(* LS Electric XG5000 project: project_7 *)
(* PLC LSPLC *)
VAR_GLOBAL
    Coil_1 : BOOL;
    CTU_R : BOOL;
    INST : CTU_DINT;
    INST1 : TON;
    Relay AT %QX0.0.1 : BOOL;
    SW_1 AT %IX0.0.1 : BOOL;
    SW_2 AT %IX0.0.2 : BOOL;
END_VAR

PROGRAM NewProgram (* task: Scan Program *)
VAR_EXTERNAL
    Coil_1 : BOOL;
    CTU_R : BOOL;
    INST : CTU_DINT;
    INST1 : TON;
    Relay : BOOL; (* AT %QX0.0.1 *)
    SW_1 : BOOL; (* AT %IX0.0.1 *)
    SW_2 : BOOL; (* AT %IX0.0.2 *)
END_VAR

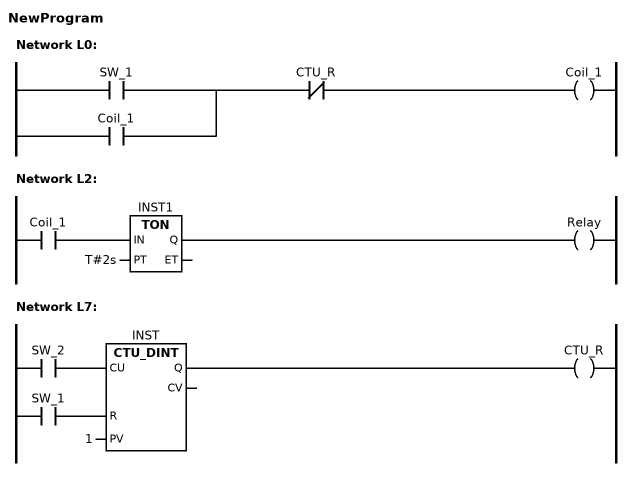
(* Rung L0 *)
Coil_1 := (SW_1 OR Coil_1) AND NOT CTU_R;
(* Rung L2 *)
INST1(IN := Coil_1, PT := T#2s);
Relay := INST1.Q;
(* Rung L7 *)
INST(CU := SW_2, R := SW_1, PV := 1);
CTU_R := INST.Q;
END_PROGRAM